(* IEC 61131-3 sources: lpmlv2022/test (part 2) *)

(* ---- TestConfigureModeTransitionCfg.st ---- *)
USING AxUnit;
USING Simatic.Ax.LPMLV2022;

NAMESPACE Simatic.Ax.LPMLV2022.Tests

    {TestFixture}
    CLASS TestConfigureModeTransitionCfg

        {Test}
        METHOD PUBLIC TestOnlyClearing
            VAR_TEMP
                result : DWORD;
            END_VAR

            ConfigureModeTransitionCfg(
                Clearing := TRUE,
                Stopped := FALSE, Starting := FALSE, Idle := FALSE, Suspended := FALSE, Execute := FALSE,
                Stopping := FALSE, Aborting := FALSE, Aborted := FALSE, Holding := FALSE, Held := FALSE,
                Unholding := FALSE, Suspending := FALSE, Unsuspending := FALSE, Resetting := FALSE,
                Completing := FALSE, Completed := FALSE,
                ModeTransitionCfg => result);

            Assert.Equal(actual := result.%X1, expected := TRUE);
            Assert.Equal(actual := result.%X2, expected := FALSE);
            // Verify expected DWORD value (bit 1 set = 2^1 = 2 = 16#02)
            Assert.Equal(actual := result, expected := DWORD#16#0000_0002);

        END_METHOD

        {Test}
        METHOD PUBLIC TestOnlyStopped
            VAR_TEMP
                result : DWORD;
            END_VAR

            ConfigureModeTransitionCfg(
                Clearing := FALSE,
                Stopped := TRUE, Starting := FALSE, Idle := FALSE, Suspended := FALSE, Execute := FALSE,
                Stopping := FALSE, Aborting := FALSE, Aborted := FALSE, Holding := FALSE, Held := FALSE,
                Unholding := FALSE, Suspending := FALSE, Unsuspending := FALSE, Resetting := FALSE,
                Completing := FALSE, Completed := FALSE,
                ModeTransitionCfg => result);

            Assert.Equal(actual := result.%X2, expected := TRUE);
            Assert.Equal(actual := result.%X1, expected := FALSE);
            // Verify expected DWORD value (bit 2 set = 2^2 = 4 = 16#04)
            Assert.Equal(actual := result, expected := DWORD#16#0000_0004);

        END_METHOD

        {Test}
        METHOD PUBLIC TestOnlyStarting
            VAR_TEMP
                result : DWORD;
            END_VAR

            ConfigureModeTransitionCfg(
                Clearing := FALSE, Stopped := FALSE,
                Starting := TRUE, Idle := FALSE, Suspended := FALSE, Execute := FALSE,
                Stopping := FALSE, Aborting := FALSE, Aborted := FALSE, Holding := FALSE, Held := FALSE,
                Unholding := FALSE, Suspending := FALSE, Unsuspending := FALSE, Resetting := FALSE,
                Completing := FALSE, Completed := FALSE,
                ModeTransitionCfg => result);

            Assert.Equal(actual := result.%X3, expected := TRUE);
            // Verify expected DWORD value (bit 3 set = 2^3 = 8 = 16#08)
            Assert.Equal(actual := result, expected := DWORD#16#0000_0008);

        END_METHOD

        {Test}
        METHOD PUBLIC TestOnlyIdle
            VAR_TEMP
                result : DWORD;
            END_VAR

            ConfigureModeTransitionCfg(
                Clearing := FALSE, Stopped := FALSE, Starting := FALSE,
                Idle := TRUE, Suspended := FALSE, Execute := FALSE,
                Stopping := FALSE, Aborting := FALSE, Aborted := FALSE, Holding := FALSE, Held := FALSE,
                Unholding := FALSE, Suspending := FALSE, Unsuspending := FALSE, Resetting := FALSE,
                Completing := FALSE, Completed := FALSE,
                ModeTransitionCfg => result);

            Assert.Equal(actual := result.%X4, expected := TRUE);
            // Verify expected DWORD value (bit 4 set = 2^4 = 16 = 16#10)
            Assert.Equal(actual := result, expected := DWORD#16#0000_0010);

        END_METHOD

        {Test}
        METHOD PUBLIC TestOnlySuspended
            VAR_TEMP
                result : DWORD;
            END_VAR

            ConfigureModeTransitionCfg(
                Clearing := FALSE, Stopped := FALSE, Starting := FALSE, Idle := FALSE,
                Suspended := TRUE, Execute := FALSE,
                Stopping := FALSE, Aborting := FALSE, Aborted := FALSE, Holding := FALSE, Held := FALSE,
                Unholding := FALSE, Suspending := FALSE, Unsuspending := FALSE, Resetting := FALSE,
                Completing := FALSE, Completed := FALSE,
                ModeTransitionCfg => result);

            Assert.Equal(actual := result.%X5, expected := TRUE);
            // Verify expected DWORD value (bit 5 set = 2^5 = 32 = 16#20)
            Assert.Equal(actual := result, expected := DWORD#16#0000_0020);

        END_METHOD

        {Test}
        METHOD PUBLIC TestOnlyExecute
            VAR_TEMP
                result : DWORD;
            END_VAR

            ConfigureModeTransitionCfg(
                Clearing := FALSE, Stopped := FALSE, Starting := FALSE, Idle := FALSE, Suspended := FALSE,
                Execute := TRUE,
                Stopping := FALSE, Aborting := FALSE, Aborted := FALSE, Holding := FALSE, Held := FALSE,
                Unholding := FALSE, Suspending := FALSE, Unsuspending := FALSE, Resetting := FALSE,
                Completing := FALSE, Completed := FALSE,
                ModeTransitionCfg => result);

            Assert.Equal(actual := result.%X6, expected := TRUE);
            // Verify expected DWORD value (bit 6 set = 2^6 = 64 = 16#40)
            Assert.Equal(actual := result, expected := DWORD#16#0000_0040);

        END_METHOD

        {Test}
        METHOD PUBLIC TestOnlyStopping
            VAR_TEMP
                result : DWORD;
            END_VAR

            ConfigureModeTransitionCfg(
                Clearing := FALSE, Stopped := FALSE, Starting := FALSE, Idle := FALSE, Suspended := FALSE, Execute := FALSE,
                Stopping := TRUE, Aborting := FALSE, Aborted := FALSE, Holding := FALSE, Held := FALSE,
                Unholding := FALSE, Suspending := FALSE, Unsuspending := FALSE, Resetting := FALSE,
                Completing := FALSE, Completed := FALSE,
                ModeTransitionCfg => result);

            Assert.Equal(actual := result.%X7, expected := TRUE);
            // Verify expected DWORD value (bit 7 set = 2^7 = 128 = 16#80)
            Assert.Equal(actual := result, expected := DWORD#16#0000_0080);

        END_METHOD

        {Test}
        METHOD PUBLIC TestOnlyAborting
            VAR_TEMP
                result : DWORD;
            END_VAR

            ConfigureModeTransitionCfg(
                Clearing := FALSE, Stopped := FALSE, Starting := FALSE, Idle := FALSE, Suspended := FALSE, Execute := FALSE,
                Stopping := FALSE, Aborting := TRUE, Aborted := FALSE, Holding := FALSE, Held := FALSE,
                Unholding := FALSE, Suspending := FALSE, Unsuspending := FALSE, Resetting := FALSE,
                Completing := FALSE, Completed := FALSE,
                ModeTransitionCfg => result);

            Assert.Equal(actual := result.%X8, expected := TRUE);
            // Verify expected DWORD value (bit 8 set = 2^8 = 256 = 16#100)
            Assert.Equal(actual := result, expected := DWORD#16#0000_0100);

        END_METHOD

        {Test}
        METHOD PUBLIC TestOnlyAborted
            VAR_TEMP
                result : DWORD;
            END_VAR

            ConfigureModeTransitionCfg(
                Clearing := FALSE, Stopped := FALSE, Starting := FALSE, Idle := FALSE, Suspended := FALSE, Execute := FALSE,
                Stopping := FALSE, Aborting := FALSE, Aborted := TRUE, Holding := FALSE, Held := FALSE,
                Unholding := FALSE, Suspending := FALSE, Unsuspending := FALSE, Resetting := FALSE,
                Completing := FALSE, Completed := FALSE,
                ModeTransitionCfg => result);

            Assert.Equal(actual := result.%X9, expected := TRUE);
            // Verify expected DWORD value (bit 9 set = 2^9 = 512 = 16#200)
            Assert.Equal(actual := result, expected := DWORD#16#0000_0200);

        END_METHOD

        {Test}
        METHOD PUBLIC TestOnlyHolding
            VAR_TEMP
                result : DWORD;
            END_VAR

            ConfigureModeTransitionCfg(
                Clearing := FALSE, Stopped := FALSE, Starting := FALSE, Idle := FALSE, Suspended := FALSE, Execute := FALSE,
                Stopping := FALSE, Aborting := FALSE, Aborted := FALSE, Holding := TRUE, Held := FALSE,
                Unholding := FALSE, Suspending := FALSE, Unsuspending := FALSE, Resetting := FALSE,
                Completing := FALSE, Completed := FALSE,
                ModeTransitionCfg => result);

            Assert.Equal(actual := result.%X10, expected := TRUE);
            // Verify expected DWORD value (bit 10 set = 2^10 = 1024 = 16#400)
            Assert.Equal(actual := result, expected := DWORD#16#0000_0400);

        END_METHOD

        {Test}
        METHOD PUBLIC TestOnlyHeld
            VAR_TEMP
                result : DWORD;
            END_VAR

            ConfigureModeTransitionCfg(
                Clearing := FALSE, Stopped := FALSE, Starting := FALSE, Idle := FALSE, Suspended := FALSE, Execute := FALSE,
                Stopping := FALSE, Aborting := FALSE, Aborted := FALSE, Holding := FALSE, Held := TRUE,
                Unholding := FALSE, Suspending := FALSE, Unsuspending := FALSE, Resetting := FALSE,
                Completing := FALSE, Completed := FALSE,
                ModeTransitionCfg => result);

            Assert.Equal(actual := result.%X11, expected := TRUE);
            // Verify expected DWORD value (bit 11 set = 2^11 = 2048 = 16#800)
            Assert.Equal(actual := result, expected := DWORD#16#0000_0800);

        END_METHOD

        {Test}
        METHOD PUBLIC TestHighOrderStates
            VAR_TEMP
                result : DWORD;
            END_VAR

            // Test Completing and Completed states (bits 16 and 17)
            ConfigureModeTransitionCfg(
                Clearing := FALSE, Stopped := FALSE, Starting := FALSE, Idle := FALSE, Suspended := FALSE, Execute := FALSE,
                Stopping := FALSE, Aborting := FALSE, Aborted := FALSE, Holding := FALSE, Held := FALSE,
                Unholding := FALSE, Suspending := FALSE, Unsuspending := FALSE, Resetting := FALSE,
                Completing := TRUE, Completed := TRUE,
                ModeTransitionCfg => result);

            Assert.Equal(actual := result.%X16, expected := TRUE);  // Completing
            Assert.Equal(actual := result.%X17, expected := TRUE);  // Completed
            // Verify expected DWORD value (bits 16+17 set = 65536+131072 = 196608 = 16#30000)
            Assert.Equal(actual := result, expected := DWORD#16#0003_0000);

        END_METHOD

        {Test}
        METHOD PUBLIC TestBasicStateTransitions
            VAR_TEMP
                result : DWORD;
            END_VAR

            // Test basic state transitions: Stopped, Starting, Idle, Execute
            ConfigureModeTransitionCfg(
                Clearing := FALSE,
                Stopped := TRUE, Starting := TRUE, Idle := TRUE, Suspended := FALSE, Execute := TRUE,
                Stopping := FALSE, Aborting := FALSE, Aborted := FALSE, Holding := FALSE, Held := FALSE,
                Unholding := FALSE, Suspending := FALSE, Unsuspending := FALSE, Resetting := FALSE,
                Completing := FALSE, Completed := FALSE,
                ModeTransitionCfg => result);

            Assert.Equal(actual := result.%X2, expected := TRUE);   // Stopped
            Assert.Equal(actual := result.%X3, expected := TRUE);   // Starting
            Assert.Equal(actual := result.%X4, expected := TRUE);   // Idle
            Assert.Equal(actual := result.%X6, expected := TRUE);   // Execute

            // Verify expected DWORD value (bits 2+3+4+6 set = 4+8+16+64 = 92 = 16#5C)
            Assert.Equal(actual := result, expected := DWORD#16#0000_005C);

        END_METHOD

        {Test}
        METHOD PUBLIC TestSuspendingStates
            VAR_TEMP
                result : DWORD;
            END_VAR

            // Test suspending-related states
            ConfigureModeTransitionCfg(
                Clearing := FALSE, Stopped := FALSE, Starting := FALSE, Idle := FALSE,
                Suspended := TRUE, Execute := FALSE,
                Stopping := FALSE, Aborting := FALSE, Aborted := FALSE, Holding := FALSE, Held := FALSE,
                Unholding := FALSE, Suspending := TRUE, Unsuspending := TRUE, Resetting := FALSE,
                Completing := FALSE, Completed := FALSE,
                ModeTransitionCfg => result);

            Assert.Equal(actual := result.%X5, expected := TRUE);   // Suspended
            Assert.Equal(actual := result.%X13, expected := TRUE);  // Suspending
            Assert.Equal(actual := result.%X14, expected := TRUE);  // Unsuspending

            // Verify expected DWORD value (bits 5+13+14 set = 32+8192+16384 = 24608 = 16#6020)
            Assert.Equal(actual := result, expected := DWORD#16#0000_6020);

        END_METHOD

        {Test}
        METHOD PUBLIC TestHoldingStates
            VAR_TEMP
                result : DWORD;
            END_VAR

            // Test holding-related states
            ConfigureModeTransitionCfg(
                Clearing := FALSE, Stopped := FALSE, Starting := FALSE, Idle := FALSE, Suspended := FALSE, Execute := FALSE,
                Stopping := FALSE, Aborting := FALSE, Aborted := FALSE,
                Holding := TRUE, Held := TRUE, Unholding := TRUE,
                Suspending := FALSE, Unsuspending := FALSE, Resetting := FALSE,
                Completing := FALSE, Completed := FALSE,
                ModeTransitionCfg => result);

            Assert.Equal(actual := result.%X10, expected := TRUE);  // Holding
            Assert.Equal(actual := result.%X11, expected := TRUE);  // Held
            Assert.Equal(actual := result.%X12, expected := TRUE);  // Unholding

            // Verify expected DWORD value (bits 10+11+12 set = 1024+2048+4096 = 7168 = 16#1C00)
            Assert.Equal(actual := result, expected := DWORD#16#0000_1C00);

        END_METHOD

        {Test}
        METHOD PUBLIC TestAbortingStates
            VAR_TEMP
                result : DWORD;
            END_VAR

            // Test aborting-related states
            ConfigureModeTransitionCfg(
                Clearing := FALSE, Stopped := FALSE, Starting := FALSE, Idle := FALSE, Suspended := FALSE, Execute := FALSE,
                Stopping := FALSE, Aborting := TRUE, Aborted := TRUE, Holding := FALSE, Held := FALSE,
                Unholding := FALSE, Suspending := FALSE, Unsuspending := FALSE, Resetting := TRUE,
                Completing := FALSE, Completed := FALSE,
                ModeTransitionCfg => result);

            Assert.Equal(actual := result.%X8, expected := TRUE);   // Aborting
            Assert.Equal(actual := result.%X9, expected := TRUE);   // Aborted
            Assert.Equal(actual := result.%X15, expected := TRUE);  // Resetting

            // Verify expected DWORD value (bits 8+9+15 set = 256+512+32768 = 33536 = 16#8300)
            Assert.Equal(actual := result, expected := DWORD#16#0000_8300);

        END_METHOD

        {Test}
        METHOD PUBLIC TestCompletingStates
            VAR_TEMP
                result : DWORD;
            END_VAR

            // Test completing-related states
            ConfigureModeTransitionCfg(
                Clearing := FALSE, Stopped := FALSE, Starting := FALSE, Idle := FALSE, Suspended := FALSE,
                Execute := TRUE,
                Stopping := FALSE, Aborting := FALSE, Aborted := FALSE, Holding := FALSE, Held := FALSE,
                Unholding := FALSE, Suspending := FALSE, Unsuspending := FALSE, Resetting := FALSE,
                Completing := TRUE, Completed := TRUE,
                ModeTransitionCfg => result);

            Assert.Equal(actual := result.%X6, expected := TRUE);   // Execute
            Assert.Equal(actual := result.%X16, expected := TRUE);  // Completing
            Assert.Equal(actual := result.%X17, expected := TRUE);  // Completed

            // Verify expected DWORD value (bits 6+16+17 set = 64+65536+131072 = 196672 = 16#30040)
            Assert.Equal(actual := result, expected := DWORD#16#0003_0040);

        END_METHOD

        {Test}
        METHOD PUBLIC TestAllStatesEnabled
            VAR_TEMP
                result : DWORD;
            END_VAR

            ConfigureModeTransitionCfg(
                Clearing := TRUE, Stopped := TRUE, Starting := TRUE, Idle := TRUE, Suspended := TRUE, Execute := TRUE,
                Stopping := TRUE, Aborting := TRUE, Aborted := TRUE, Holding := TRUE, Held := TRUE,
                Unholding := TRUE, Suspending := TRUE, Unsuspending := TRUE, Resetting := TRUE,
                Completing := TRUE, Completed := TRUE,
                ModeTransitionCfg => result);

            // Verify all configured bits are set
            Assert.Equal(actual := result.%X1, expected := TRUE);   // Clearing
            Assert.Equal(actual := result.%X2, expected := TRUE);   // Stopped
            Assert.Equal(actual := result.%X3, expected := TRUE);   // Starting
            Assert.Equal(actual := result.%X4, expected := TRUE);   // Idle
            Assert.Equal(actual := result.%X5, expected := TRUE);   // Suspended
            Assert.Equal(actual := result.%X6, expected := TRUE);   // Execute
            Assert.Equal(actual := result.%X7, expected := TRUE);   // Stopping
            Assert.Equal(actual := result.%X8, expected := TRUE);   // Aborting
            Assert.Equal(actual := result.%X9, expected := TRUE);   // Aborted
            Assert.Equal(actual := result.%X10, expected := TRUE);  // Holding
            Assert.Equal(actual := result.%X11, expected := TRUE);  // Held
            Assert.Equal(actual := result.%X12, expected := TRUE);  // Unholding
            Assert.Equal(actual := result.%X13, expected := TRUE);  // Suspending
            Assert.Equal(actual := result.%X14, expected := TRUE);  // Unsuspending
            Assert.Equal(actual := result.%X15, expected := TRUE);  // Resetting
            Assert.Equal(actual := result.%X16, expected := TRUE);  // Completing
            Assert.Equal(actual := result.%X17, expected := TRUE);  // Completed

            // Verify expected DWORD value (all configured bits 1-17 set)
            // bits 1-17 = 2+4+8+16+32+64+128+256+512+1024+2048+4096+8192+16384+32768+65536+131072 = 262142 = 16#3FFFE
            Assert.Equal(actual := result, expected := DWORD#16#0003_FFFE);

        END_METHOD

        {Test}
        METHOD PUBLIC TestAllStatesDisabled
            VAR_TEMP
                result : DWORD;
            END_VAR

            ConfigureModeTransitionCfg(
                Clearing := FALSE, Stopped := FALSE, Starting := FALSE, Idle := FALSE, Suspended := FALSE, Execute := FALSE,
                Stopping := FALSE, Aborting := FALSE, Aborted := FALSE, Holding := FALSE, Held := FALSE,
                Unholding := FALSE, Suspending := FALSE, Unsuspending := FALSE, Resetting := FALSE,
                Completing := FALSE, Completed := FALSE,
                ModeTransitionCfg => result);

            // Verify all configured bits are FALSE
            Assert.Equal(actual := result.%X1, expected := FALSE);
            Assert.Equal(actual := result.%X2, expected := FALSE);
            Assert.Equal(actual := result.%X3, expected := FALSE);
            Assert.Equal(actual := result.%X17, expected := FALSE);

            // Verify expected DWORD value (no bits set = 0)
            Assert.Equal(actual := result, expected := DWORD#16#0000_0000);

        END_METHOD

        {Test}
        METHOD PUBLIC TestUnusedBitsRemainZero
            VAR_TEMP
                result : DWORD;
            END_VAR

            // Test with all configurable states enabled
            ConfigureModeTransitionCfg(
                Clearing := TRUE, Stopped := TRUE, Starting := TRUE, Idle := TRUE, Suspended := TRUE, Execute := TRUE,
                Stopping := TRUE, Aborting := TRUE, Aborted := TRUE, Holding := TRUE, Held := TRUE,
                Unholding := TRUE, Suspending := TRUE, Unsuspending := TRUE, Resetting := TRUE,
                Completing := TRUE, Completed := TRUE,
                ModeTransitionCfg => result);

            // Test that unused bits remain 0
            Assert.Equal(actual := result.%X0, expected := FALSE);   // Unused
            Assert.Equal(actual := result.%X18, expected := FALSE);  // Unused
            Assert.Equal(actual := result.%X19, expected := FALSE);  // Unused
            Assert.Equal(actual := result.%X20, expected := FALSE);  // Unused
            Assert.Equal(actual := result.%X25, expected := FALSE);  // Unused
            Assert.Equal(actual := result.%X31, expected := FALSE);  // Unused (MSB)

        END_METHOD

        {Test}
        METHOD PUBLIC TestBitMappingVerification
            VAR_TEMP
                result : DWORD;
            END_VAR

            // Test specific bit mappings for key states

            // Test Clearing -> bit 1
            ConfigureModeTransitionCfg(
                Clearing := TRUE,
                Stopped := FALSE, Starting := FALSE, Idle := FALSE, Suspended := FALSE, Execute := FALSE,
                Stopping := FALSE, Aborting := FALSE, Aborted := FALSE, Holding := FALSE, Held := FALSE,
                Unholding := FALSE, Suspending := FALSE, Unsuspending := FALSE, Resetting := FALSE,
                Completing := FALSE, Completed := FALSE,
                ModeTransitionCfg => result);
            Assert.Equal(actual := result.%X1, expected := TRUE);
            Assert.Equal(actual := result, expected := DWORD#16#0000_0002);

            // Test Resetting -> bit 15
            ConfigureModeTransitionCfg(
                Clearing := FALSE, Stopped := FALSE, Starting := FALSE, Idle := FALSE, Suspended := FALSE, Execute := FALSE,
                Stopping := FALSE, Aborting := FALSE, Aborted := FALSE, Holding := FALSE, Held := FALSE,
                Unholding := FALSE, Suspending := FALSE, Unsuspending := FALSE,
                Resetting := TRUE,
                Completing := FALSE, Completed := FALSE,
                ModeTransitionCfg => result);
            Assert.Equal(actual := result.%X15, expected := TRUE);
            Assert.Equal(actual := result, expected := DWORD#16#0000_8000);

        END_METHOD

        {Test}
        METHOD PUBLIC TestSequentialLowOrderBits
            VAR_TEMP
                result : DWORD;
            END_VAR

            // Test first 8 states to verify sequential bit mapping
            ConfigureModeTransitionCfg(
                Clearing := TRUE, Stopped := TRUE, Starting := TRUE, Idle := TRUE,
                Suspended := TRUE, Execute := TRUE, Stopping := TRUE, Aborting := TRUE,
                Aborted := FALSE, Holding := FALSE, Held := FALSE,
                Unholding := FALSE, Suspending := FALSE, Unsuspending := FALSE, Resetting := FALSE,
                Completing := FALSE, Completed := FALSE,
                ModeTransitionCfg => result);

            Assert.Equal(actual := result.%X1, expected := TRUE);   // Clearing -> bit 1
            Assert.Equal(actual := result.%X2, expected := TRUE);   // Stopped -> bit 2
            Assert.Equal(actual := result.%X3, expected := TRUE);   // Starting -> bit 3
            Assert.Equal(actual := result.%X4, expected := TRUE);   // Idle -> bit 4
            Assert.Equal(actual := result.%X5, expected := TRUE);   // Suspended -> bit 5
            Assert.Equal(actual := result.%X6, expected := TRUE);   // Execute -> bit 6
            Assert.Equal(actual := result.%X7, expected := TRUE);   // Stopping -> bit 7
            Assert.Equal(actual := result.%X8, expected := TRUE);   // Aborting -> bit 8
            Assert.Equal(actual := result.%X9, expected := FALSE);  // Aborted -> bit 9 (should be false)

            // Verify expected DWORD value (bits 1-8 set = 2+4+8+16+32+64+128+256 = 510 = 16#1FE)
            Assert.Equal(actual := result, expected := DWORD#16#0000_01FE);

        END_METHOD

        {Test}
        METHOD PUBLIC TestAlternatingPattern
            VAR_TEMP
                result : DWORD;
            END_VAR

            // Test alternating pattern of states
            ConfigureModeTransitionCfg(
                Clearing := TRUE, Stopped := FALSE, Starting := TRUE, Idle := FALSE,
                Suspended := TRUE, Execute := FALSE, Stopping := TRUE, Aborting := FALSE,
                Aborted := TRUE, Holding := FALSE, Held := TRUE, Unholding := FALSE,
                Suspending := TRUE, Unsuspending := FALSE, Resetting := TRUE,
                Completing := FALSE, Completed := TRUE,
                ModeTransitionCfg => result);

            // Verify alternating pattern
            Assert.Equal(actual := result.%X1, expected := TRUE);   // Clearing
            Assert.Equal(actual := result.%X2, expected := FALSE);  // Stopped
            Assert.Equal(actual := result.%X3, expected := TRUE);   // Starting
            Assert.Equal(actual := result.%X4, expected := FALSE);  // Idle
            Assert.Equal(actual := result.%X17, expected := TRUE);  // Completed
            Assert.Equal(actual := result.%X16, expected := FALSE); // Completing

            // Verify alternating DWORD pattern for bits 1-17
            // Pattern: 10101010101010101 (binary) = 0x2AAAA in hex
            Assert.Equal(actual := result, expected := DWORD#16#0002_AAAA);

        END_METHOD

        {Test}
        METHOD PUBLIC TestCriticalStateTransitions
            VAR_TEMP
                result : DWORD;
            END_VAR

            // Test critical states that typically need mode transitions
            ConfigureModeTransitionCfg(
                Clearing := TRUE,   // After abort/error
                Stopped := TRUE,    // Initial state
                Starting := FALSE, Idle := TRUE,     // Normal operation
                Suspended := FALSE, Execute := FALSE,
                Stopping := TRUE,   // Controlled shutdown
                Aborting := TRUE, Aborted := TRUE,   // Emergency states
                Holding := FALSE, Held := FALSE, Unholding := FALSE,
                Suspending := FALSE, Unsuspending := FALSE,
                Resetting := TRUE,  // Recovery
                Completing := FALSE, Completed := FALSE,
                ModeTransitionCfg => result);

            Assert.Equal(actual := result.%X1, expected := TRUE);   // Clearing
            Assert.Equal(actual := result.%X2, expected := TRUE);   // Stopped
            Assert.Equal(actual := result.%X4, expected := TRUE);   // Idle
            Assert.Equal(actual := result.%X7, expected := TRUE);   // Stopping
            Assert.Equal(actual := result.%X8, expected := TRUE);   // Aborting
            Assert.Equal(actual := result.%X9, expected := TRUE);   // Aborted
            Assert.Equal(actual := result.%X15, expected := TRUE);  // Resetting

            // Verify expected DWORD value (bits 1+2+4+7+8+9+15 set)
            // = 2+4+16+128+256+512+32768 = 33686 = 16#8396
            Assert.Equal(actual := result, expected := DWORD#16#0000_8396);

        END_METHOD

    END_CLASS

END_NAMESPACE

(* ---- TestStacklight.st ---- *)
USING AxUnit;
USING Simatic.Ax.LPMLV2022;

NAMESPACE Simatic.Ax.LPMLV2022.Tests

    {TestFixture}
    CLASS TestStacklight
        VAR
            stacklight : Stacklight;
        END_VAR

        {Test}
        METHOD PUBLIC TestStateExecute_NormalOperation
            VAR_TEMP
                expectedStacklight : DWORD;
            END_VAR

            // Test Execute state with normal operation (no material issues)
            stacklight.StateCurrent := State#EXECUTE;
            stacklight.starvedUpstream := FALSE;
            stacklight.blockedDownstream := FALSE;
            stacklight.materialLow := FALSE;
            stacklight.materialExhausted := FALSE;
            stacklight();

            // Verify individual outputs
            Assert.Equal(actual := stacklight.redSolid, expected := FALSE);
            Assert.Equal(actual := stacklight.redFlashing, expected := FALSE);
            Assert.Equal(actual := stacklight.amberSolid, expected := FALSE);
            Assert.Equal(actual := stacklight.amberFlashing, expected := FALSE);
            Assert.Equal(actual := stacklight.blueSolid, expected := FALSE);
            Assert.Equal(actual := stacklight.blueFlashing, expected := FALSE);
            Assert.Equal(actual := stacklight.greenSolid, expected := TRUE);      // Running - Green Solid
            Assert.Equal(actual := stacklight.greenFlashing, expected := FALSE);
            Assert.Equal(actual := stacklight.hornFlashing, expected := FALSE);

            // Verify DWORD output (bit 6 set = 2^6 = 64 = 16#40)
            Assert.Equal(actual := stacklight.StacklightStatus, expected := DWORD#16#0000_0040);

        END_METHOD

        {Test}
        METHOD PUBLIC TestStateExecute_WithMaterialLow
            VAR_TEMP
                expectedStacklight : DWORD;
            END_VAR

            // Test Execute state with low material
            stacklight.StateCurrent := State#EXECUTE;
            stacklight.starvedUpstream := FALSE;
            stacklight.blockedDownstream := FALSE;
            stacklight.materialLow := TRUE;
            stacklight.materialExhausted := FALSE;
            stacklight();

            // Verify outputs
            Assert.Equal(actual := stacklight.greenSolid, expected := TRUE);      // Running
            Assert.Equal(actual := stacklight.blueFlashing, expected := TRUE);    // Low material
            Assert.Equal(actual := stacklight.redSolid, expected := FALSE);
            Assert.Equal(actual := stacklight.hornFlashing, expected := FALSE);

            // Verify DWORD output (bits 5+6 set = 32+64 = 96 = 16#60)
            Assert.Equal(actual := stacklight.StacklightStatus, expected := DWORD#16#0000_0060);

        END_METHOD

        {Test}
        METHOD PUBLIC TestStateIdle_ReadyToStart
            VAR_TEMP
                expectedStacklight : DWORD;
            END_VAR

            // Test Idle state (ready to start)
            stacklight.StateCurrent := State#IDLE;
            stacklight.starvedUpstream := FALSE;
            stacklight.blockedDownstream := FALSE;
            stacklight.materialLow := FALSE;
            stacklight.materialExhausted := FALSE;
            stacklight();

            // Verify outputs
            Assert.Equal(actual := stacklight.greenFlashing, expected := TRUE);   // Ready to start
            Assert.Equal(actual := stacklight.greenSolid, expected := FALSE);
            Assert.Equal(actual := stacklight.blueFlashing, expected := FALSE);
            Assert.Equal(actual := stacklight.hornFlashing, expected := FALSE);

            // Verify DWORD output (bit 7 set = 2^7 = 128 = 16#80)
            Assert.Equal(actual := stacklight.StacklightStatus, expected := DWORD#16#0000_0080);

        END_METHOD

        {Test}
        METHOD PUBLIC TestStateStarting_WithHorn
            VAR_TEMP
                expectedStacklight : DWORD;
            END_VAR

            // Test Starting state
            stacklight.StateCurrent := State#STARTING;
            stacklight.starvedUpstream := FALSE;
            stacklight.blockedDownstream := FALSE;
            stacklight.materialLow := FALSE;
            stacklight.materialExhausted := FALSE;
            stacklight();

            // Verify outputs
            Assert.Equal(actual := stacklight.greenSolid, expected := TRUE);      // Running
            Assert.Equal(actual := stacklight.hornFlashing, expected := TRUE);    // Starting/Restarting
            Assert.Equal(actual := stacklight.greenFlashing, expected := FALSE);
            Assert.Equal(actual := stacklight.blueFlashing, expected := FALSE);

            // Verify DWORD output (bits 6+9 set = 64+512 = 576 = 16#240)
            Assert.Equal(actual := stacklight.StacklightStatus, expected := DWORD#16#0000_0240);

        END_METHOD

        {Test}
        METHOD PUBLIC TestStateAborting_AbnormalStop
            VAR_TEMP
                expectedStacklight : DWORD;
            END_VAR

            // Test Aborting state (abnormal stop)
            stacklight.StateCurrent := State#ABORTING;
            stacklight.starvedUpstream := FALSE;
            stacklight.blockedDownstream := FALSE;
            stacklight.materialLow := FALSE;
            stacklight.materialExhausted := FALSE;
            stacklight();

            // Verify outputs
            Assert.Equal(actual := stacklight.redFlashing, expected := TRUE);     // Abnormal stop
            Assert.Equal(actual := stacklight.redSolid, expected := FALSE);
            Assert.Equal(actual := stacklight.greenSolid, expected := FALSE);
            Assert.Equal(actual := stacklight.blueFlashing, expected := FALSE);

            // Verify DWORD output (bit 1 set = 2^1 = 2 = 16#02)
            Assert.Equal(actual := stacklight.StacklightStatus, expected := DWORD#16#0000_0002);

        END_METHOD

        {Test}
        METHOD PUBLIC TestStateStopped_ControlledStop
            VAR_TEMP
                expectedStacklight : DWORD;
            END_VAR

            // Test Stopped state (controlled stop)
            stacklight.StateCurrent := State#STOPPED;
            stacklight.starvedUpstream := FALSE;
            stacklight.blockedDownstream := FALSE;
            stacklight.materialLow := FALSE;
            stacklight.materialExhausted := FALSE;
            stacklight();

            // Verify outputs
            Assert.Equal(actual := stacklight.redSolid, expected := TRUE);        // Controlled stop
            Assert.Equal(actual := stacklight.redFlashing, expected := FALSE);
            Assert.Equal(actual := stacklight.greenSolid, expected := FALSE);
            Assert.Equal(actual := stacklight.blueFlashing, expected := FALSE);

            // Verify DWORD output (bit 0 set = 2^0 = 1 = 16#01)
            Assert.Equal(actual := stacklight.StacklightStatus, expected := DWORD#16#0000_0001);

        END_METHOD

        {Test}
        METHOD PUBLIC TestStateSuspended_StarvedUpstream
            VAR_TEMP
                expectedStacklight : DWORD;
            END_VAR

            // Test Suspended state with starved upstream
            stacklight.StateCurrent := State#SUSPENDED;
            stacklight.starvedUpstream := TRUE;
            stacklight.blockedDownstream := FALSE;
            stacklight.materialLow := FALSE;
            stacklight.materialExhausted := FALSE;
            stacklight();

            // Verify outputs
            Assert.Equal(actual := stacklight.amberFlashing, expected := TRUE);   // Starved upstream
            Assert.Equal(actual := stacklight.amberSolid, expected := FALSE);
            Assert.Equal(actual := stacklight.blueFlashing, expected := FALSE);
            Assert.Equal(actual := stacklight.greenSolid, expected := FALSE);

            // Verify DWORD output (bit 3 set = 2^3 = 8 = 16#08)
            Assert.Equal(actual := stacklight.StacklightStatus, expected := DWORD#16#0000_0008);

        END_METHOD

        {Test}
        METHOD PUBLIC TestStateSuspended_BlockedDownstream
            VAR_TEMP
                expectedStacklight : DWORD;
            END_VAR

            // Test Suspended state with blocked downstream
            stacklight.StateCurrent := State#SUSPENDED;
            stacklight.starvedUpstream := FALSE;
            stacklight.blockedDownstream := TRUE;
            stacklight.materialLow := FALSE;
            stacklight.materialExhausted := FALSE;
            stacklight();

            // Verify outputs
            Assert.Equal(actual := stacklight.amberSolid, expected := TRUE);      // Blocked downstream
            Assert.Equal(actual := stacklight.amberFlashing, expected := FALSE);
            Assert.Equal(actual := stacklight.blueFlashing, expected := FALSE);

            // Verify DWORD output (bit 2 set = 2^2 = 4 = 16#04)
            Assert.Equal(actual := stacklight.StacklightStatus, expected := DWORD#16#0000_0004);

        END_METHOD

        {Test}
        METHOD PUBLIC TestStateHeld_MaterialExhausted
            VAR_TEMP
                expectedStacklight : DWORD;
            END_VAR

            // Test Held state with material exhausted
            stacklight.StateCurrent := State#HELD;
            stacklight.starvedUpstream := FALSE;
            stacklight.blockedDownstream := FALSE;
            stacklight.materialLow := FALSE;
            stacklight.materialExhausted := TRUE;
            stacklight();

            // Verify outputs
            Assert.Equal(actual := stacklight.blueSolid, expected := TRUE);       // Material exhausted
            Assert.Equal(actual := stacklight.blueFlashing, expected := FALSE);
            Assert.Equal(actual := stacklight.greenSolid, expected := FALSE);

            // Verify DWORD output (bit 4 set = 2^4 = 16 = 16#10)
            Assert.Equal(actual := stacklight.StacklightStatus, expected := DWORD#16#0000_0010);

        END_METHOD

        {Test}
        METHOD PUBLIC TestStateUnholding_RestartingWithHorn
            VAR_TEMP
                expectedStacklight : DWORD;
            END_VAR

            // Test Unholding state (restarting with horn)
            stacklight.StateCurrent := State#UNHOLDING;
            stacklight.starvedUpstream := FALSE;
            stacklight.blockedDownstream := FALSE;
            stacklight.materialLow := FALSE;
            stacklight.materialExhausted := FALSE;
            stacklight();

            // Verify outputs
            Assert.Equal(actual := stacklight.greenSolid, expected := TRUE);      // Running
            Assert.Equal(actual := stacklight.hornFlashing, expected := TRUE);    // Restarting
            Assert.Equal(actual := stacklight.blueFlashing, expected := FALSE);

            // Verify DWORD output (bits 6+9 set = 64+512 = 576 = 16#240)
            Assert.Equal(actual := stacklight.StacklightStatus, expected := DWORD#16#0000_0240);

        END_METHOD

        {Test}
        METHOD PUBLIC TestComplexScenario_SuspendedWithAllConditions
            VAR_TEMP
                expectedStacklight : DWORD;
            END_VAR

            // Test complex scenario: Suspended with all conditions active
            stacklight.StateCurrent := State#SUSPENDED;
            stacklight.starvedUpstream := TRUE;
            stacklight.blockedDownstream := TRUE;
            stacklight.materialLow := TRUE;
            stacklight.materialExhausted := FALSE;
            stacklight();

            // Verify outputs
            Assert.Equal(actual := stacklight.amberFlashing, expected := TRUE);   // Starved upstream
            Assert.Equal(actual := stacklight.amberSolid, expected := TRUE);      // Blocked downstream
            Assert.Equal(actual := stacklight.blueFlashing, expected := TRUE);    // Low material
            Assert.Equal(actual := stacklight.blueSolid, expected := FALSE);
            Assert.Equal(actual := stacklight.greenSolid, expected := FALSE);

            // Verify DWORD output (bits 2+3+5 set = 4+8+32 = 44 = 16#2C)
            Assert.Equal(actual := stacklight.StacklightStatus, expected := DWORD#16#0000_002C);

        END_METHOD

        {Test}
        METHOD PUBLIC TestStateCompleting_RunningWithMaterial
            VAR_TEMP
                expectedStacklight : DWORD;
            END_VAR

            // Test Completing state
            stacklight.StateCurrent := State#COMPLETING;
            stacklight.starvedUpstream := FALSE;
            stacklight.blockedDownstream := FALSE;
            stacklight.materialLow := TRUE;
            stacklight.materialExhausted := FALSE;
            stacklight();

            // Verify outputs
            Assert.Equal(actual := stacklight.greenSolid, expected := TRUE);      // Running
            Assert.Equal(actual := stacklight.blueFlashing, expected := TRUE);    // Low material
            Assert.Equal(actual := stacklight.hornFlashing, expected := FALSE);

            // Verify DWORD output (bits 5+6 set = 32+64 = 96 = 16#60)
            Assert.Equal(actual := stacklight.StacklightStatus, expected := DWORD#16#0000_0060);

        END_METHOD

        {Test}
        METHOD PUBLIC TestAllAbnormalStates
            VAR_TEMP
                expectedStacklight : DWORD;
            END_VAR

            // Test all abnormal stop states (should show red flashing)

            // Test Aborting
            stacklight.StateCurrent := State#ABORTING;
            stacklight.starvedUpstream := FALSE;
            stacklight.blockedDownstream := FALSE;
            stacklight.materialLow := FALSE;
            stacklight.materialExhausted := FALSE;
            stacklight();
            Assert.Equal(actual := stacklight.redFlashing, expected := TRUE);
            Assert.Equal(actual := stacklight.redSolid, expected := FALSE);

            // Test Aborted
            stacklight.StateCurrent := State#ABORTED;
            stacklight();
            Assert.Equal(actual := stacklight.redFlashing, expected := TRUE);
            Assert.Equal(actual := stacklight.redSolid, expected := FALSE);

            // Test Clearing
            stacklight.StateCurrent := State#CLEARING;
            stacklight();
            Assert.Equal(actual := stacklight.redFlashing, expected := TRUE);
            Assert.Equal(actual := stacklight.redSolid, expected := FALSE);

        END_METHOD

        {Test}
        METHOD PUBLIC TestAllControlledStopStates
            VAR_TEMP
                expectedStacklight : DWORD;
            END_VAR

            // Test all controlled stop states (should show red solid)

            // Test Completed
            stacklight.StateCurrent := State#COMPLETED;
            stacklight.starvedUpstream := FALSE;
            stacklight.blockedDownstream := FALSE;
            stacklight.materialLow := FALSE;
            stacklight.materialExhausted := FALSE;
            stacklight();
            Assert.Equal(actual := stacklight.redSolid, expected := TRUE);
            Assert.Equal(actual := stacklight.redFlashing, expected := FALSE);

            // Test Resetting
            stacklight.StateCurrent := State#RESETTING;
            stacklight();
            Assert.Equal(actual := stacklight.redSolid, expected := TRUE);
            Assert.Equal(actual := stacklight.redFlashing, expected := FALSE);

            // Test Stopping
            stacklight.StateCurrent := State#STOPPING;
            stacklight();
            Assert.Equal(actual := stacklight.redSolid, expected := TRUE);
            Assert.Equal(actual := stacklight.redFlashing, expected := FALSE);

            // Test Stopped
            stacklight.StateCurrent := State#STOPPED;
            stacklight();
            Assert.Equal(actual := stacklight.redSolid, expected := TRUE);
            Assert.Equal(actual := stacklight.redFlashing, expected := FALSE);

        END_METHOD

        {Test}
        METHOD PUBLIC TestAllRunningStates
            VAR_TEMP
                expectedStacklight : DWORD;
            END_VAR

            // Test all running states (should show green solid)

            // Test Execute
            stacklight.StateCurrent := State#EXECUTE;
            stacklight.starvedUpstream := FALSE;
            stacklight.blockedDownstream := FALSE;
            stacklight.materialLow := FALSE;
            stacklight.materialExhausted := FALSE;
            stacklight();
            Assert.Equal(actual := stacklight.greenSolid, expected := TRUE);
            Assert.Equal(actual := stacklight.greenFlashing, expected := FALSE);

            // Test Starting
            stacklight.StateCurrent := State#STARTING;
            stacklight();
            Assert.Equal(actual := stacklight.greenSolid, expected := TRUE);
            Assert.Equal(actual := stacklight.hornFlashing, expected := TRUE);

            // Test Completing
            stacklight.StateCurrent := State#COMPLETING;
            stacklight();
            Assert.Equal(actual := stacklight.greenSolid, expected := TRUE);
            Assert.Equal(actual := stacklight.hornFlashing, expected := FALSE);

            // Test Unholding
            stacklight.StateCurrent := State#UNHOLDING;
            stacklight();
            Assert.Equal(actual := stacklight.greenSolid, expected := TRUE);
            Assert.Equal(actual := stacklight.hornFlashing, expected := TRUE);

            // Test Unsuspending
            stacklight.StateCurrent := State#UNSUSPENDING;
            stacklight();
            Assert.Equal(actual := stacklight.greenSolid, expected := TRUE);
            Assert.Equal(actual := stacklight.hornFlashing, expected := TRUE);

        END_METHOD

        {Test}
        METHOD PUBLIC TestHornFlashingStates
            VAR_TEMP
                expectedStacklight : DWORD;
            END_VAR

            // Test all states that should trigger horn flashing
            stacklight.starvedUpstream := FALSE;
            stacklight.blockedDownstream := FALSE;
            stacklight.materialLow := FALSE;
            stacklight.materialExhausted := FALSE;

            // Starting
            stacklight.StateCurrent := State#STARTING;
            stacklight();
            Assert.Equal(actual := stacklight.hornFlashing, expected := TRUE);

            // Unholding
            stacklight.StateCurrent := State#UNHOLDING;
            stacklight();
            Assert.Equal(actual := stacklight.hornFlashing, expected := TRUE);

            // Unsuspending
            stacklight.StateCurrent := State#UNSUSPENDING;
            stacklight();
            Assert.Equal(actual := stacklight.hornFlashing, expected := TRUE);

            // Other states should not have horn
            stacklight.StateCurrent := State#EXECUTE;
            stacklight();
            Assert.Equal(actual := stacklight.hornFlashing, expected := FALSE);

        END_METHOD

        {Test}
        METHOD PUBLIC TestMaterialConditionsInVariousStates
            VAR_TEMP
                expectedStacklight : DWORD;
            END_VAR

            // Test material conditions in states where they should be active

            // Low material in Execute state
            stacklight.StateCurrent := State#EXECUTE;
            stacklight.starvedUpstream := FALSE;
            stacklight.blockedDownstream := FALSE;
            stacklight.materialLow := TRUE;
            stacklight.materialExhausted := FALSE;
            stacklight();
            Assert.Equal(actual := stacklight.blueFlashing, expected := TRUE);
            Assert.Equal(actual := stacklight.blueSolid, expected := FALSE);

            // Material exhausted in Held state
            stacklight.StateCurrent := State#HELD;
            stacklight.materialLow := FALSE;
            stacklight.materialExhausted := TRUE;
            stacklight();
            Assert.Equal(actual := stacklight.blueSolid, expected := TRUE);
            Assert.Equal(actual := stacklight.blueFlashing, expected := FALSE);

            // Low material should not affect Holding state blue solid logic
            stacklight.StateCurrent := State#HOLDING;
            stacklight.materialLow := TRUE;
            stacklight.materialExhausted := FALSE;
            stacklight();
            Assert.Equal(actual := stacklight.blueSolid, expected := FALSE);
            Assert.Equal(actual := stacklight.blueFlashing, expected := FALSE);

        END_METHOD

        {Test}
        METHOD PUBLIC TestUndefinedState
            VAR_TEMP
                expectedStacklight : DWORD;
            END_VAR

            // Test undefined state (should reset all outputs)
            stacklight.StateCurrent := State#UNDEFINED;
            stacklight.starvedUpstream := TRUE;
            stacklight.blockedDownstream := TRUE;
            stacklight.materialLow := TRUE;
            stacklight.materialExhausted := TRUE;
            stacklight();

            // All outputs should be FALSE for undefined state
            Assert.Equal(actual := stacklight.redSolid, expected := FALSE);
            Assert.Equal(actual := stacklight.redFlashing, expected := FALSE);
            Assert.Equal(actual := stacklight.amberSolid, expected := FALSE);
            Assert.Equal(actual := stacklight.amberFlashing, expected := FALSE);
            Assert.Equal(actual := stacklight.blueSolid, expected := FALSE);
            Assert.Equal(actual := stacklight.blueFlashing, expected := FALSE);
            Assert.Equal(actual := stacklight.greenSolid, expected := FALSE);
            Assert.Equal(actual := stacklight.greenFlashing, expected := FALSE);
            Assert.Equal(actual := stacklight.hornFlashing, expected := FALSE);

            // Verify DWORD output (no bits set = 0)
            Assert.Equal(actual := stacklight.StacklightStatus, expected := DWORD#16#0000_0000);

        END_METHOD

        {Test}
        METHOD PUBLIC TestStacklightBitMapping
            VAR_TEMP
                expectedStacklight : DWORD;
            END_VAR

            // Test that individual outputs correctly map to DWORD bits

            // Test red solid (bit 0)
            stacklight.StateCurrent := State#STOPPED;
            stacklight.starvedUpstream := FALSE;
            stacklight.blockedDownstream := FALSE;
            stacklight.materialLow := FALSE;
            stacklight.materialExhausted := FALSE;
            stacklight();
            Assert.Equal(actual := stacklight.StacklightStatus.%X0, expected := TRUE);
            Assert.Equal(actual := stacklight.redSolid, expected := TRUE);

            // Test green flashing (bit 7)
            stacklight.StateCurrent := State#IDLE;
            stacklight();
            Assert.Equal(actual := stacklight.StacklightStatus.%X7, expected := TRUE);
            Assert.Equal(actual := stacklight.greenFlashing, expected := TRUE);

            // Test horn flashing (bit 9)
            stacklight.StateCurrent := State#STARTING;
            stacklight();
            Assert.Equal(actual := stacklight.StacklightStatus.%X9, expected := TRUE);
            Assert.Equal(actual := stacklight.hornFlashing, expected := TRUE);

        END_METHOD

        {Test}
        METHOD PUBLIC TestUnusedStacklightBits
            VAR_TEMP
                expectedStacklight : DWORD;
            END_VAR

            // Test that unused bits in the DWORD remain zero
            stacklight.StateCurrent := State#STARTING;
            stacklight.starvedUpstream := TRUE;
            stacklight.blockedDownstream := TRUE;
            stacklight.materialLow := TRUE;
            stacklight.materialExhausted := TRUE;
            stacklight();

            // Verify that unused bits are FALSE
            Assert.Equal(actual := stacklight.StacklightStatus.%X8, expected := FALSE);   // Unused bit 8
            Assert.Equal(actual := stacklight.StacklightStatus.%X10, expected := FALSE);  // Unused bit 10
            Assert.Equal(actual := stacklight.StacklightStatus.%X15, expected := FALSE);  // Unused bit 15
            Assert.Equal(actual := stacklight.StacklightStatus.%X31, expected := FALSE);  // Unused bit 31 (MSB)

        END_METHOD

        {Test}
        METHOD PUBLIC TestANSICompliance_TableVerification
            VAR_TEMP
                expectedStacklight : DWORD;
            END_VAR

            // Verify ANSI compliance based on the comment table in the source code

            // Abnormal Stop: Aborting, Clearing, Aborted -> Red Flashing
            stacklight.StateCurrent := State#ABORTING;
            stacklight.starvedUpstream := FALSE;
            stacklight.blockedDownstream := FALSE;
            stacklight.materialLow := FALSE;
            stacklight.materialExhausted := FALSE;
            stacklight();
            Assert.Equal(actual := stacklight.redFlashing, expected := TRUE);

            // Controlled Stop: Completed, Stopped, Stopping, Resetting -> Red Solid
            stacklight.StateCurrent := State#COMPLETED;
            stacklight();
            Assert.Equal(actual := stacklight.redSolid, expected := TRUE);

            // Ready to Start: Idle -> Green Flashing
            stacklight.StateCurrent := State#IDLE;
            stacklight();
            Assert.Equal(actual := stacklight.greenFlashing, expected := TRUE);

            // Running: Starting, Execute, Completing, Unholding, Unsuspending -> Green Solid
            stacklight.StateCurrent := State#EXECUTE;
            stacklight();
            Assert.Equal(actual := stacklight.greenSolid, expected := TRUE);

            // Starting/Restarting: Starting, Unholding, Unsuspending -> Horn
            stacklight.StateCurrent := State#STARTING;
            stacklight();
            Assert.Equal(actual := stacklight.hornFlashing, expected := TRUE);

        END_METHOD

        {Test}
        METHOD PUBLIC TestSequentialStateCalls
            VAR_TEMP
                expectedStacklight : DWORD;
            END_VAR

            // Test that multiple sequential calls work correctly (function block behavior)

            // First call - Execute state
            stacklight.StateCurrent := State#EXECUTE;
            stacklight.starvedUpstream := FALSE;
            stacklight.blockedDownstream := FALSE;
            stacklight.materialLow := FALSE;
            stacklight.materialExhausted := FALSE;
            stacklight();
            Assert.Equal(actual := stacklight.greenSolid, expected := TRUE);
            Assert.Equal(actual := stacklight.redSolid, expected := FALSE);

            // Second call - change to Stopped state
            stacklight.StateCurrent := State#STOPPED;
            stacklight();
            Assert.Equal(actual := stacklight.redSolid, expected := TRUE);
            Assert.Equal(actual := stacklight.greenSolid, expected := FALSE);

            // Third call - change to Idle state
            stacklight.StateCurrent := State#IDLE;
            stacklight();
            Assert.Equal(actual := stacklight.greenFlashing, expected := TRUE);
            Assert.Equal(actual := stacklight.redSolid, expected := FALSE);
            Assert.Equal(actual := stacklight.greenSolid, expected := FALSE);

        END_METHOD

        {Test}
        METHOD PUBLIC TestSuspending
            VAR_TEMP
                expectedStacklight : DWORD;
            END_VAR

            stacklight.StateCurrent := State#SUSPENDING;
            stacklight.starvedUpstream := TRUE;
            stacklight.blockedDownstream := TRUE;
            stacklight.materialLow := TRUE;
            stacklight.materialExhausted := FALSE;
            stacklight();

            Assert.Equal(actual := stacklight.amberFlashing, expected := TRUE);
            Assert.Equal(actual := stacklight.amberSolid, expected := TRUE);
            Assert.Equal(actual := stacklight.blueFlashing, expected := TRUE);
            // Verify DWORD output (bits 2,3,5 set = 16#2C
            Assert.Equal(actual := stacklight.StacklightStatus, expected := DWORD#16#0000_002C);

        END_METHOD

    END_CLASS

END_NAMESPACE

(* ---- TestUnitModeStateManager.st ---- *)
USING AxUnit;
USING Simatic.Ax.LPMLV2022;

NAMESPACE Simatic.Ax.LPMLV2022.Tests

    {TestFixture}
    CLASS TestStopNotAllowedInStop
        VAR
            unitModeManager : UnitModeStateManager;
        END_VAR

        {Test}
        METHOD PUBLIC TestStopNotAllowedInStop_RisingEdge
            VAR_TEMP
                i : UINT;
            END_VAR

            FOR i := 0 TO UINT#10 DO
                unitModeManager();
            END_FOR;

            unitModeManager.CntrlCmd := Command#START;
            unitModeManager.CmdChangeRequest := TRUE;

            FOR i := 0 TO UINT#10 DO
                unitModeManager();
            END_FOR;

            Assert.Equal(actual := unitModeManager.cntrlCmdNotAllowed, expected := TRUE);
            Assert.Equal(actual := unitModeManager.diagnostics.buffer[0].message, expected := BYTE#16#84); //  MSG_CMD_NOT_ALLOWED : Byte := BYTE#16#84;

        END_METHOD
    END_CLASS

    {TestFixture}
    CLASS TestCmdNotAllowedInResetting
        VAR
            unitModeManager : UnitModeStateManager;
        END_VAR

        {Test}
        METHOD PUBLIC TestStopNotAllowedInStop_RisingEdge
            VAR_TEMP
                i : UINT;
            END_VAR

            unitModeManager();  // First cycle

            // Test rising edge detection for Reset command
            unitModeManager.CntrlCmd := Command#RESET;
            unitModeManager();

            // Rising edge - should trigger command
            unitModeManager.CmdChangeRequest := TRUE;
            FOR i := 0 TO UINT#10 DO
                unitModeManager();
            END_FOR;

            unitModeManager.CmdChangeRequest := FALSE;
            FOR i := 0 TO UINT#10 DO
                unitModeManager();
            END_FOR;

            unitModeManager.CntrlCmd := Command#START;
            unitModeManager.CmdChangeRequest := TRUE;
            // CMD_STARET in RESETTING not allowed
            FOR i := 0 TO UINT#10 DO
                unitModeManager();
            END_FOR;
            Assert.Equal(actual := unitModeManager.cntrlCmdNotAllowed, expected := TRUE);
            Assert.Equal(actual := unitModeManager.diagnostics.buffer[1].message, expected := BYTE#16#84); //  MSG_CMD_NOT_ALLOWED : Byte := BYTE#16#84;

        END_METHOD
    END_CLASS

    {TestFixture}
    CLASS TestExecuteCompleteTransition
        VAR
            unitModeManager : UnitModeStateManager;
        END_VAR

        {Test}
        METHOD PUBLIC TestExecuteCompletingTransition
            VAR_TEMP
                i : UINT;
                disabled : DWORD;
            END_VAR

            ConfigureDisabledStatesCfg(Completing := TRUE,  DisabledStatesCfg => disabled);
            unitModeManager.config.DisabledStatesCfg[1] := disabled;
            unitModeManager();  // First cycle

            unitModeManager.UnitMode := Mode#PRODUCTION;
            unitModeManager.UnitModeChangeRequest := TRUE;
            FOR i := 0 TO UINT#10 DO
                unitModeManager();
            END_FOR;
            unitModeManager.UnitModeChangeRequest := FALSE;
            Assert.Equal(actual := unitModeManager.UnitModeCurrent, expected := Mode#PRODUCTION);

            // Test rising edge detection for Reset command
            unitModeManager.CntrlCmd := Command#RESET;
            unitModeManager();

            // Rising edge - should trigger command
            unitModeManager.CmdChangeRequest := TRUE;
            FOR i := 0 TO UINT#10 DO
                unitModeManager();
            END_FOR;

            unitModeManager.CmdChangeRequest := FALSE;
            unitModeManager.SC := TRUE;
            FOR i := 0 TO UINT#10 DO
                unitModeManager();
            END_FOR;

            unitModeManager.CntrlCmd := Command#START;
            unitModeManager.CmdChangeRequest := TRUE;
            unitModeManager.SC := FALSE;
            FOR i := 0 TO UINT#10 DO
                unitModeManager();
            END_FOR;

            unitModeManager.CmdChangeRequest := FALSE;
            unitModeManager.SC := TRUE;
            FOR i := 0 TO UINT#10 DO
                unitModeManager();
            END_FOR;

            unitModeManager.CntrlCmd := Command#COMPLETE;
            unitModeManager.CmdChangeRequest := TRUE;
            unitModeManager.SC := FALSE;
            FOR i := 0 TO UINT#10 DO
                unitModeManager();
            END_FOR;
            Assert.Equal(actual := unitModeManager.StateCurrent, expected := State#COMPLETED);

        END_METHOD
    END_CLASS

    {TestFixture}
    CLASS TestExecuteHoldTransition
        VAR
            unitModeManager : UnitModeStateManager;
        END_VAR

        {Test}
        METHOD PUBLIC TestExecuteHoldingTransition
            VAR_TEMP
                i : UINT;
                disabled : DWORD;
            END_VAR

            ConfigureDisabledStatesCfg(Holding := TRUE,  DisabledStatesCfg => disabled);
            unitModeManager.config.DisabledStatesCfg[1] := disabled;
            unitModeManager();  // First cycle

            unitModeManager.UnitMode := Mode#PRODUCTION;
            unitModeManager.UnitModeChangeRequest := TRUE;
            FOR i := 0 TO UINT#10 DO
                unitModeManager();
            END_FOR;
            unitModeManager.UnitModeChangeRequest := FALSE;
            Assert.Equal(actual := unitModeManager.UnitModeCurrent, expected := Mode#PRODUCTION);

            // Test rising edge detection for Reset command
            unitModeManager.CntrlCmd := Command#RESET;
            unitModeManager();

            // Rising edge - should trigger command
            unitModeManager.CmdChangeRequest := TRUE;
            FOR i := 0 TO UINT#10 DO
                unitModeManager();
            END_FOR;

            unitModeManager.CmdChangeRequest := FALSE;
            unitModeManager.SC := TRUE;
            FOR i := 0 TO UINT#10 DO
                unitModeManager();
            END_FOR;

            unitModeManager.CntrlCmd := Command#START;
            unitModeManager.CmdChangeRequest := TRUE;
            unitModeManager.SC := FALSE;
            FOR i := 0 TO UINT#10 DO
                unitModeManager();
            END_FOR;

            unitModeManager.CmdChangeRequest := FALSE;
            unitModeManager.SC := TRUE;
            FOR i := 0 TO UINT#10 DO
                unitModeManager();
            END_FOR;

            unitModeManager.CntrlCmd := Command#HOLD;
            unitModeManager.CmdChangeRequest := TRUE;
            unitModeManager.SC := FALSE;
            FOR i := 0 TO UINT#10 DO
                unitModeManager();
            END_FOR;
            Assert.Equal(actual := unitModeManager.StateCurrent, expected := State#HELD);

        END_METHOD
    END_CLASS

    {TestFixture}
    CLASS TestExecuteSuspendedTransition
        VAR
            unitModeManager : UnitModeStateManager;
        END_VAR

        {Test}
        METHOD PUBLIC TestExecuteSuspendedTransition_Test
            VAR_TEMP
                i : UINT;
                disabled : DWORD;
            END_VAR

            ConfigureDisabledStatesCfg(Suspending := TRUE,  DisabledStatesCfg => disabled);
            unitModeManager.config.DisabledStatesCfg[1] := disabled;
            unitModeManager();  // First cycle

            unitModeManager.UnitMode := Mode#PRODUCTION;
            unitModeManager.UnitModeChangeRequest := TRUE;
            FOR i := 0 TO UINT#10 DO
                unitModeManager();
            END_FOR;
            unitModeManager.UnitModeChangeRequest := FALSE;
            Assert.Equal(actual := unitModeManager.UnitModeCurrent, expected := Mode#PRODUCTION);

            // Test rising edge detection for Reset command
            unitModeManager.CntrlCmd := Command#RESET;
            unitModeManager();

            // Rising edge - should trigger command
            unitModeManager.CmdChangeRequest := TRUE;
            FOR i := 0 TO UINT#10 DO
                unitModeManager();
            END_FOR;

            unitModeManager.CmdChangeRequest := FALSE;
            unitModeManager.SC := TRUE;
            FOR i := 0 TO UINT#10 DO
                unitModeManager();
            END_FOR;

            unitModeManager.CntrlCmd := Command#START;
            unitModeManager.CmdChangeRequest := TRUE;
            unitModeManager.SC := FALSE;
            FOR i := 0 TO UINT#10 DO
                unitModeManager();
            END_FOR;

            unitModeManager.CmdChangeRequest := FALSE;
            unitModeManager.SC := TRUE;
            FOR i := 0 TO UINT#10 DO
                unitModeManager();
            END_FOR;

            unitModeManager.CntrlCmd := Command#SUSPEND;
            unitModeManager.CmdChangeRequest := TRUE;
            unitModeManager.SC := FALSE;
            FOR i := 0 TO UINT#10 DO
                unitModeManager();
            END_FOR;
            Assert.Equal(actual := unitModeManager.StateCurrent, expected := State#SUSPENDED);

        END_METHOD
    END_CLASS

    {TestFixture}
    CLASS TestHoldAfterCompleted
        VAR
            unitModeManager : UnitModeStateManager;
        END_VAR

        {Test}
        METHOD PUBLIC TestHoldAfterCompleted_Test
            VAR_TEMP
                i : UINT;
                holdCfg : DWORD;
            END_VAR

            ConfigureHoldCmdCfg(Completed := TRUE,  holdCmdCfg => holdCfg);
            unitModeManager.config.holdCmdCfg := holdCfg;
            unitModeManager();  // First cycle

            unitModeManager.UnitMode := Mode#PRODUCTION;
            unitModeManager.UnitModeChangeRequest := TRUE;
            FOR i := 0 TO UINT#10 DO
                unitModeManager();
            END_FOR;
            unitModeManager.UnitModeChangeRequest := FALSE;
            Assert.Equal(actual := unitModeManager.UnitModeCurrent, expected := Mode#PRODUCTION);

            // Test rising edge detection for Reset command
            unitModeManager.CntrlCmd := Command#RESET;
            unitModeManager();

            // Rising edge - should trigger command
            unitModeManager.CmdChangeRequest := TRUE;
            FOR i := 0 TO UINT#10 DO
                unitModeManager();
            END_FOR;

            unitModeManager.CmdChangeRequest := FALSE;
            unitModeManager.SC := TRUE;
            FOR i := 0 TO UINT#10 DO
                unitModeManager();
            END_FOR;

            unitModeManager.CntrlCmd := Command#START;
            unitModeManager.CmdChangeRequest := TRUE;
            unitModeManager.SC := FALSE;
            FOR i := 0 TO UINT#10 DO
                unitModeManager();
            END_FOR;

            unitModeManager.CmdChangeRequest := FALSE;
            unitModeManager.SC := TRUE;
            FOR i := 0 TO UINT#10 DO
                unitModeManager();
            END_FOR;

            unitModeManager.CntrlCmd := Command#COMPLETE;
            unitModeManager.CmdChangeRequest := TRUE;
            unitModeManager.SC := FALSE;
            FOR i := 0 TO UINT#10 DO
                unitModeManager();
            END_FOR;

            unitModeManager.CmdChangeRequest := FALSE;
            unitModeManager.SC := TRUE;
            FOR i := 0 TO UINT#10 DO
                unitModeManager();
            END_FOR;

            unitModeManager.CntrlCmd := Command#HOLD;
            unitModeManager.CmdChangeRequest := TRUE;
            unitModeManager.SC := FALSE;
            FOR i := 0 TO UINT#10 DO
                unitModeManager();
            END_FOR;
            Assert.Equal(actual := unitModeManager.StateCurrent, expected := State#HOLDING);

        END_METHOD
    END_CLASS
END_NAMESPACE
